// TIA Portal V16 export
// export: Created 2024-11-21T10:48:16.144789Z, ExportSetting WithDefaults, DisplayName Totally Integrated Automation Portal, DisplayVersion V16 Update 6, DisplayName TIA Portal Version Control Interface, DisplayVersion V16 Update 2, DisplayName TIA Portal Openness, DisplayVersion V16 Update 6, DisplayName STEP 7 Professional, DisplayVersion V16 Update 6, DisplayName STEP 7 Safety, DisplayVersion V16, DisplayName WinCC Advanced / Unified PC, DisplayVersion V16 Update 6
FUNCTION_BLOCK "FB_INDUCTA"   // FB10024, LAD
{ S7_Optimized_Access := 'TRUE' }
VERSION : 0.1
// stored: AutoNumber false, IsIECCheckEnabled false, IsRetainMemResEnabled false, MemoryReserve 100, SetENOAutomatically false, UDAEnableTagReadback false
   VAR_INPUT
      iENB : Bool;
      iALM_RST : Bool;
   END_VAR
   VAR_OUTPUT
      oHeater : Bool;
      oPower : Word;
   END_VAR
   VAR_IN_OUT
      ioData : "UDT_INDUCTA";
   END_VAR
   VAR
      _HeatingTime : Time;
      HeatingTON { S7_SetPoint := 'True'} : IEC_TIMER;
      EmergencyTON { S7_SetPoint := 'True'} : IEC_TIMER;
   END_VAR
   VAR CONSTANT
      MAX_TIME : Time := T#10s;
   END_VAR
   VAR_TEMP   // added for the SCL form of the ladder/FBD networks
      _w1 : Bool;
   END_VAR
BEGIN

REGION Network 1: Operating mode
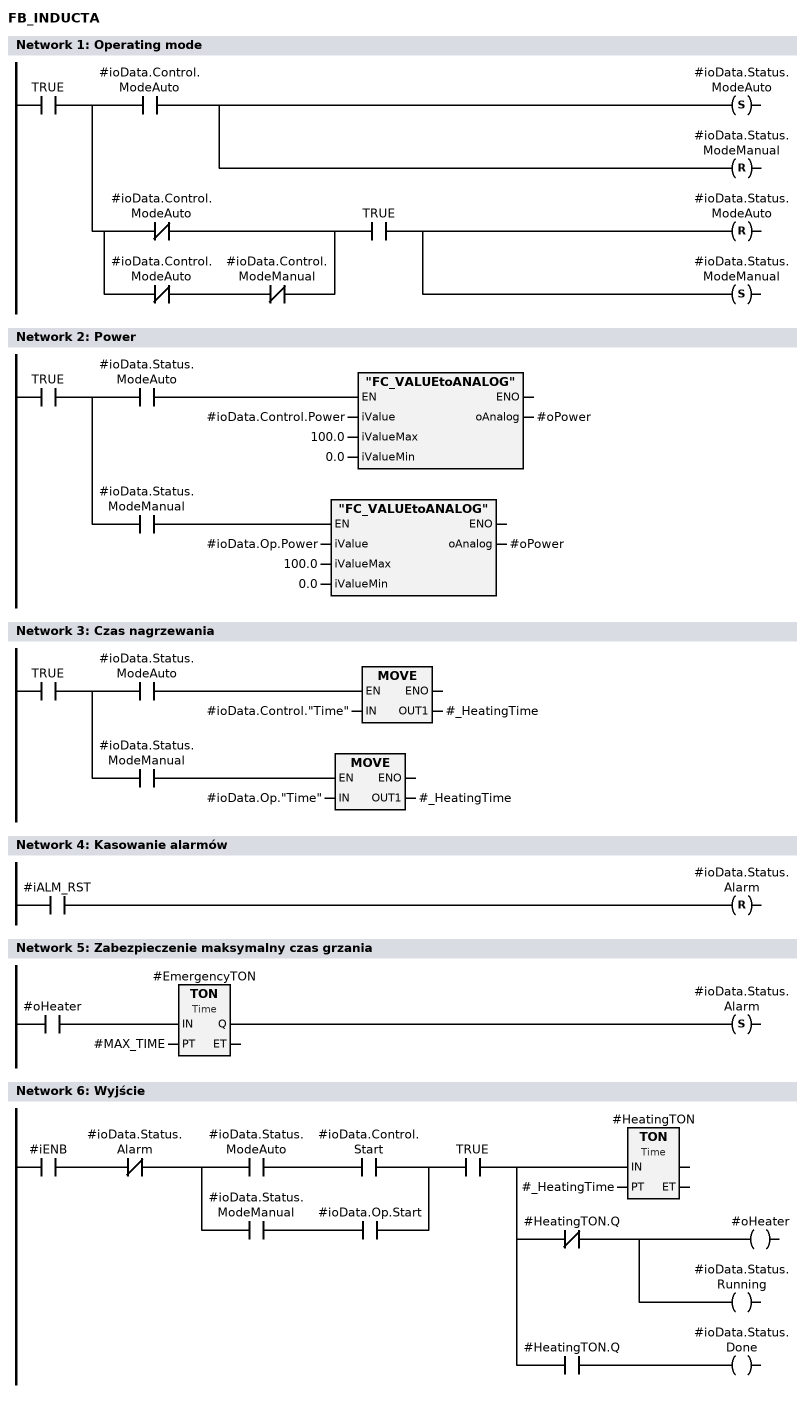
   RUNG wire#powerrail
      Contact( TRUE )
      wire#w1
      Contact( #ioData.Control.ModeAuto )
      wire#w2
      S_Coil( #ioData.Status.ModeAuto )
   END_RUNG
   RUNG wire#w2
      R_Coil( #ioData.Status.ModeManual )
   END_RUNG
   RUNG wire#w1
      I_Contact( #ioData.Control.ModeAuto )
      wire#w3
      Contact( TRUE )
      wire#w4
      R_Coil( #ioData.Status.ModeAuto )
   END_RUNG
   RUNG wire#w1
      I_Contact( #ioData.Control.ModeAuto )
      I_Contact( #ioData.Control.ModeManual )
   END_RUNG wire#w3
   RUNG wire#w4
      S_Coil( #ioData.Status.ModeManual )
   END_RUNG
   // the same network as SCL:
   IF TRUE AND #ioData.Control.ModeAuto THEN
       #ioData.Status.ModeAuto := TRUE;
       #ioData.Status.ModeManual := FALSE;
   END_IF;
   IF TRUE AND (NOT #ioData.Control.ModeAuto OR (NOT #ioData.Control.ModeAuto AND NOT #ioData.Control.ModeManual)) AND TRUE THEN
       #ioData.Status.ModeAuto := FALSE;
       #ioData.Status.ModeManual := TRUE;
   END_IF;
END_REGION

REGION Network 2: Power
   RUNG wire#powerrail
      Contact( TRUE )
      wire#w1
      Contact( #ioData.Status.ModeAuto )
      "FC_VALUEtoANALOG"(iValue := #ioData.Control.Power, iValueMax := 100.0, iValueMin := 0.0, oAnalog => #oPower)
   END_RUNG
   RUNG wire#w1
      Contact( #ioData.Status.ModeManual )
      "FC_VALUEtoANALOG"(iValue := #ioData.Op.Power, iValueMax := 100.0, iValueMin := 0.0, oAnalog => #oPower)
   END_RUNG
   // the same network as SCL:
   IF TRUE AND #ioData.Status.ModeAuto THEN
       "FC_VALUEtoANALOG"(iValue := #ioData.Control.Power, iValueMax := 100.0, iValueMin := 0.0, oAnalog => #oPower);
   END_IF;
   IF TRUE AND #ioData.Status.ModeManual THEN
       "FC_VALUEtoANALOG"(iValue := #ioData.Op.Power, iValueMax := 100.0, iValueMin := 0.0, oAnalog => #oPower);
   END_IF;
END_REGION

REGION Network 3: Czas nagrzewania
   RUNG wire#powerrail
      Contact( TRUE )
      wire#w1
      Contact( #ioData.Status.ModeAuto )
      Move(in := #ioData.Control."Time", out1 => #_HeatingTime)
   END_RUNG
   RUNG wire#w1
      Contact( #ioData.Status.ModeManual )
      Move(in := #ioData.Op."Time", out1 => #_HeatingTime)
   END_RUNG
   // the same network as SCL:
   IF TRUE AND #ioData.Status.ModeAuto THEN #_HeatingTime := #ioData.Control."Time"; END_IF;
   IF TRUE AND #ioData.Status.ModeManual THEN #_HeatingTime := #ioData.Op."Time"; END_IF;
END_REGION

REGION Network 4: Kasowanie alarmów
   RUNG wire#powerrail
      Contact( #iALM_RST )
      R_Coil( #ioData.Status.Alarm )
   END_RUNG
   // the same network as SCL:
   IF #iALM_RST THEN #ioData.Status.Alarm := FALSE; END_IF;
END_REGION

REGION Network 5: Zabezpieczenie maksymalny czas grzania
   RUNG wire#powerrail
      Contact( #oHeater )
      { S7_Templates := "time_type := Time" } #EmergencyTON.TON(pt := #MAX_TIME, et =>)
      S_Coil( #ioData.Status.Alarm )
   END_RUNG
   // the same network as SCL:
   #EmergencyTON.TON(IN := #oHeater, PT := #MAX_TIME);
   IF #EmergencyTON.Q THEN #ioData.Status.Alarm := TRUE; END_IF;
END_REGION

REGION Network 6: Wyjście
   RUNG wire#powerrail
      Contact( #iENB )
      I_Contact( #ioData.Status.Alarm )
      wire#w1
      Contact( #ioData.Status.ModeAuto )
      Contact( #ioData.Control.Start )
      wire#w2
      Contact( TRUE )
      wire#w3
      { S7_Templates := "time_type := Time" } #HeatingTON.TON(pt := #_HeatingTime, et =>)
   END_RUNG
   RUNG wire#w1
      Contact( #ioData.Status.ModeManual )
      Contact( #ioData.Op.Start )
   END_RUNG wire#w2
   RUNG wire#w3
      I_Contact( #HeatingTON.Q )
      wire#w4
      Coil( #oHeater )
   END_RUNG
   RUNG wire#w4
      Coil( #ioData.Status.Running )
   END_RUNG
   RUNG wire#w3
      Contact( #HeatingTON.Q )
      Coil( #ioData.Status.Done )
   END_RUNG
   // the same network as SCL:
   #_w1 := #iENB AND NOT #ioData.Status.Alarm AND ((#ioData.Status.ModeAuto AND #ioData.Control.Start) OR (#ioData.Status.ModeManual AND #ioData.Op.Start)) AND TRUE;
   #HeatingTON.TON(IN := #_w1, PT := #_HeatingTime);
   #oHeater := #_w1 AND NOT #HeatingTON.Q;
   #ioData.Status.Running := #oHeater;
   #ioData.Status.Done := #_w1 AND #HeatingTON.Q;
END_REGION
END_FUNCTION_BLOCK
